(* PLC project Tc2_Math.LMOD Demo, tc3-libraries-kb TwinCAT 3.1 *)
(* stored: creationDateTime 2026-05-10T10:00:00, modificationDateTime 2026-05-10T10:00:00 *)

PROGRAM P_Demo_LMOD
  VAR
    rResult : LREAL;  (* LMOD 的返回值 *)
    bRun : BOOL;  (* 触发一次调用 *)
  END_VAR

            // ============================================================
// Tc2_Math.LMOD 演示程序（FUNCTION）
// ============================================================
// 验证步骤：
//   1. 引用 Tc2_Math
//   2. 编译 + 登录
//   3. 强制 bRun := TRUE 一个周期
//   4. 在线监视 rResult 应为 40.56
// ============================================================

IF bRun THEN
    rResult := LMOD(400.56, 360.0);
    bRun := FALSE;
END_IF;

          
END_PROGRAM
